ABB RAPID module: TCP_mtip_tool2_nest.mod

MODULE TCP_mtip_tool2_nest
	! Points are read in order of declaration.
  ! Please do not change the order of points!

  LOCAL PERS robtarget pTCP_Point1:=[[476.736,-1007.055,598.7921],[0.0205076038837433,0.993922829627991,-0.107828430831432,-0.00835722871124744],[-1,-3,-1,1],[9E+09,9E+09,9E+09,9E+09,9E+09,9E+09]];
	LOCAL PERS robtarget pTCP_Point2:=[[86.48785,-1134.158,494.0105],[0.0957460775971413,-0.95799994468689,0.108406148850918,-0.24762250483036],[-1,-2,-2,1],[9E+09,9E+09,9E+09,9E+09,9E+09,9E+09]];
	LOCAL PERS robtarget pTCP_Point3:=[[233.8687,-1349.098,493.1813],[0.226485848426819,-0.961280584335327,0.0719815120100975,-0.139508008956909],[-1,-2,-1,1],[9E+09,9E+09,9E+09,9E+09,9E+09,9E+09]];
	LOCAL PERS robtarget pTCP_Point4:=[[744.6267,-1118.038,538.6064],[0.052165050059557,-0.979517698287964,0.0213511344045401,0.193308115005493],[-1,-3,-1,1],[9E+09,9E+09,9E+09,9E+09,9E+09,9E+09]];
	LOCAL PERS robtarget pTCP_Point5:=[[741.9869,-783.5103,497.9237],[0.170718938112259,0.965741097927094,0.00822694506496191,-0.195272788405418],[-1,-3,-1,1],[9E+09,9E+09,9E+09,9E+09,9E+09,9E+09]];
	LOCAL PERS robtarget pTCP_Point6:=[[640.0015,-644.7266,465.5243],[0.241356879472733,0.937005221843719,0.182814046740532,-0.174204230308533],[-1,-3,-1,1],[9E+09,9E+09,9E+09,9E+09,9E+09,9E+09]];
	LOCAL PERS robtarget pTCP_Point7:=[[352.0727,-888.8716,577.2051],[0.057993907481432,0.889545083045959,-0.440285533666611,0.107214458286762],[-1,-2,-1,1],[9E+09,9E+09,9E+09,9E+09,9E+09,9E+09]];
	LOCAL PERS robtarget pTCP_Point8:=[[89.37123,-966.447,499.8433],[0.158505216240883,-0.63147646188736,0.732228577136993,-0.199887067079544],[-1,-2,-1,1],[9E+09,9E+09,9E+09,9E+09,9E+09,9E+09]];

ENDMODULE
